{attribute 'qualified_only'}
VAR_GLOBAL
    nScans : UDINT;
    bTimerDone : BOOL;
END_VAR
VAR_GLOBAL CONSTANT
    MAX_STEP : DINT := 7;
END_VAR

(* stored: Version 1.1.0.1, ProductVersion 3.1.4024.12
   GVL GVL_Main: Id {5f1c2d9e-0a6b-4c11-9d3e-7a1b2c3d4e30} *)
